FUNCTION Matrix_Shrink : Bool
VAR_IN_OUT CONSTANT
	M_From : Matrix;
END_VAR
VAR_IN_OUT
	M_To : Matrix;
END_VAR
VAR_INPUT
	Row : UINT;
	Col : UINT;
END_VAR


VAR
	Ri : UINT;
	Ci : UINT;
END_VAR

IF M_From.Length <= 1 THEN
	Matrix_Shrink := FALSE;
	RETURN;
END_IF

IF M_To.Rows <> MAX(1,M_From.Rows-1) OR M_To.Cols <> MAX(1,M_From.Cols-1) THEN
	Matrix_Shrink := FALSE;
	RETURN;
END_IF

IF Row >= M_From.Rows OR Col >= M_From.Cols THEN
	Matrix_Shrink := FALSE;
	RETURN;
END_IF

Matrix_Shrink := TRUE;

FOR Ri := 0 TO M_To.Rows-1 DO
	FOR Ci := 0 TO M_To.Cols-1 DO
		M_To.SetRC(Ri,Ci,M_From.GetRC(Ri + BOOL_TO_UINT(Ri >= Row AND M_From.Rows <> M_To.Rows),Ci + BOOL_TO_UINT(Ci >= Col AND M_From.Cols <> M_To.Cols)));
	END_FOR
END_FOR

END_FUNCTION

(* stored: Version 1.1.0.1, ProductVersion 3.1.4024.9
   POU Matrix_Shrink: Id {d21782ed-5125-47a2-8d89-29ac4702d315}, SpecialFunc None *)
